Fanuc KAREL source: kt00004.KL

-- PROVISIONAL review KL for V770-1; original PC SHA256 fb4241101d99c4d77dd1d9f95b1ee1a20eecf738c7a6699711e84a1fcf728dc3
-- Incomplete behavior may be omitted. Consult companion uncertainty JSON. Do not deploy.
PROGRAM KT00004
%NOLOCKGROUP
VAR
  I1 : INTEGER
  R2 : REAL
  OUT : REAL
BEGIN
  -- UNRESOLVED_PC offsets 5-16; opcodes 2E,23
  -- UNRESOLVED_PC offsets 21-32; opcodes 2E,23
  -- UNRESOLVED_PC offsets 37-58; opcodes 21,21,29,64,69,23
  -- UNRESOLVED_PC offsets 63-67; opcodes 7F
END KT00004
